INTERFACE I_RecipesManager

PROPERTY Active : REFERENCE TO BOOL
GET
END_GET
END_PROPERTY

PROPERTY Busy : REFERENCE TO BOOL
GET
END_GET
END_PROPERTY

PROPERTY Error : REFERENCE TO BOOL
GET
END_GET
END_PROPERTY

PROPERTY ErrorID : REFERENCE TO DWORD
GET
END_GET
END_PROPERTY

PROPERTY LastResult : REFERENCE TO E_RecipesManagerReturns
GET
END_GET
END_PROPERTY

METHOD MR_Abort : BOOL
VAR_INPUT
END_VAR
END_METHOD

METHOD MR_Backup : BOOL
VAR_INPUT
	sRecipesDefinition		: STRING;
	sRecipeName				: STRING;
	sBackupStoragePath		: STRING;
END_VAR
END_METHOD

METHOD MR_Create : BOOL
VAR_INPUT
	sRecipesDefinition : STRING;
	sRecipeName : STRING;
END_VAR
END_METHOD

METHOD MR_GetRecipesNames : BOOL
VAR_INPUT
	sRecipesDefinition : STRING;
END_VAR
END_METHOD

METHOD MR_GetVariablesNames : BOOL
VAR_INPUT
	sRecipesDefinition	: STRING;
	sRecipeName : STRING;
END_VAR
END_METHOD

METHOD MR_GetVariableValues : BOOL
VAR_INPUT
	sRecipesDefinition	: STRING;
	sRecipeName : STRING;
END_VAR
END_METHOD

METHOD MR_Init : BOOL
VAR_INPUT
END_VAR
END_METHOD

METHOD MR_Load : BOOL
VAR_INPUT
	sRecipesDefinition : STRING;
	sRecipeName : STRING;
END_VAR
END_METHOD

METHOD MR_LoadAndWritte : BOOL
VAR_INPUT
	sRecipesDefinition : STRING;
	sRecipeName : STRING;
END_VAR
END_METHOD

METHOD MR_Read : BOOL
VAR_INPUT
	sRecipesDefinition : STRING;
	sRecipeName : STRING;
END_VAR
END_METHOD

METHOD MR_ReadAndSave : BOOL
VAR_INPUT
	sRecipesDefinition : STRING;
	sRecipeName : STRING;
END_VAR
END_METHOD

METHOD MR_Reload : BOOL
VAR_INPUT
	sRecipeName : STRING;
	sRecipesDefinition : STRING;
END_VAR
END_METHOD

METHOD MR_ReloadExternal : BOOL
VAR_INPUT
	sRecipeName 			: STRING;
	sRecipesDefinition 		: STRING;
	sBackupStoragePath		: STRING;
END_VAR
END_METHOD

METHOD MR_Remove : BOOL
VAR_INPUT
	sRecipesDefinition : STRING;
	sRecipeName : STRING;
END_VAR
END_METHOD

METHOD MR_Restore : BOOL
VAR_INPUT
	sRecipesDefinition		: STRING;
	sRecipeName				: STRING;
	sBackupStoragePath		: STRING;
END_VAR
END_METHOD

METHOD MR_Save : BOOL
VAR_INPUT
	sRecipesDefinition : STRING;
	sRecipeName : STRING;
END_VAR
END_METHOD

METHOD MR_Writte : BOOL
VAR_INPUT
	sRecipesDefinition : STRING;
	sRecipeName : STRING;
END_VAR
END_METHOD

PROPERTY RecipeCount : REFERENCE TO USINT
GET
END_GET
END_PROPERTY

PROPERTY RecipesDefinition : REFERENCE TO STRING
GET
END_GET
END_PROPERTY

PROPERTY RecipesNames : REFERENCE TO ARRAY [0..iMAX_NUMBER_OF_RECIPES-1] OF STRING;
GET
END_GET
END_PROPERTY

PROPERTY RecipeValues : REFERENCE TO ARRAY [0..iMAX_NUMBER_OF_VARIABLES_IN_RECIPES-1] OF STRING
//PROPERTY RecipeValues : ARRAY [0..iMAX_NUMBER_OF_VARIABLES_IN_RECIPES-1] OF STRING(iMAX_RECIPE_NAME_LENGTH)
GET
END_GET
END_PROPERTY

PROPERTY RecipeValuesAdr : REFERENCE TO ARRAY [0..iMAX_NUMBER_OF_VARIABLES_IN_RECIPES-1] OF PVOID
GET
END_GET
END_PROPERTY

PROPERTY State : REFERENCE TO E_RecipesManagerState
GET
END_GET
END_PROPERTY

END_INTERFACE

(* stored: Version 1.1.0.1, ProductVersion 3.1.4024.12
   Itf I_RecipesManager: Id {7057ab11-af6e-493b-a220-bacdaa49dd59}
   Property Active: Id {bde34ffa-12f4-441f-bfba-71bea6fd0582}
   Get Get: Id {a452c6a0-c1af-48e5-8757-18e3cb39c475}
   Property Busy: Id {2dbc07eb-4c85-4755-acbe-ca1801cb3f83}
   Get Get: Id {d26ab1c0-6b9d-49af-bbbd-0b54b6950fb7}
   Property Error: Id {ec370076-02c1-427f-a7ce-cb62e257789d}
   Get Get: Id {a9ce79e2-c27c-447c-998e-74b99fc5c116}
   Property ErrorID: Id {03b3d0ee-1c04-4bd9-b50d-78faf2801a0d}
   Get Get: Id {ea298f4c-66d0-461e-b068-87476e613f9d}
   Property LastResult: Id {55507853-eb3f-47b7-b0e1-64c1557b8964}
   Get Get: Id {18c11fad-d0e3-4436-bbad-db091799d30a}
   Method MR_Abort: Id {43f4a9d7-ae84-4930-8a83-d7c761d7d38d}
   Method MR_Backup: Id {350fc49e-7a42-4963-bc6d-f348542a3a23}
   Method MR_Create: Id {b5dff985-0c90-4514-93bd-d89e0ee3d55c}
   Method MR_GetRecipesNames: Id {6ce1affd-3f1a-4148-8497-bf69ebefc106}
   Method MR_GetVariablesNames: Id {09bd1110-0d7f-4454-b702-d9613ede0d46}
   Method MR_GetVariableValues: Id {56bd768d-00f4-4b37-a666-dca3d11247b0}
   Method MR_Init: Id {8c99939b-3aa8-430b-922d-c6a8def04fc5}
   Method MR_Load: Id {33dd0eef-0d22-4d14-91e9-fb84e2d2b2bb}
   Method MR_LoadAndWritte: Id {3a1f24e4-f3cb-4c1b-8476-9940286f8a7d}
   Method MR_Read: Id {0dcbd69b-957a-410e-87c7-32a8393e30da}
   Method MR_ReadAndSave: Id {f38a0646-f35f-4d4b-ae1f-4a651c3f1bf6}
   Method MR_Reload: Id {ab64d9cf-1188-48f3-88e6-3c7e32af5756}
   Method MR_ReloadExternal: Id {9d321bef-5019-41e9-9b83-3d92834843d9}
   Method MR_Remove: Id {8dd2a9ab-d7bb-43e1-b8ef-ca690b7e82c2}
   Method MR_Restore: Id {d0caff79-8d4e-44d4-a4da-fb4758229a0d}
   Method MR_Save: Id {d3c65dfa-ba19-4fce-964e-891e5e86a4d5}
   Method MR_Writte: Id {85beb7bb-768a-41c1-8d96-3cc9c0197717}
   Property RecipeCount: Id {8dea1c76-d94a-47af-afde-307495d64bbd}
   Get Get: Id {7cf6118e-a992-464a-9529-638210286c15}
   Property RecipesDefinition: Id {e79cb469-7eac-4b13-8c1a-aa1b5864dc10}
   Get Get: Id {1526d50a-e62d-4506-8ff8-46a658cc24a1}
   Property RecipesNames: Id {9fcb0d35-8fca-4128-b9b3-5fa195d7a347}
   Get Get: Id {62bdd0db-e7e7-41b3-8ae6-5ce4905d2572}
   Property RecipeValues: Id {9de71902-b78e-4d2c-b2e3-a5aa7a35b706}
   Get Get: Id {9a8113d5-a3d5-425f-b71c-feb9dcebd1fb}
   Property RecipeValuesAdr: Id {5097eb6d-4186-47c4-a693-6e422f4a2757}
   Get Get: Id {aab75d28-cfc1-471a-bf58-198081c94f52}
   Property State: Id {d0bbd71e-19aa-499f-a925-0a93e89e0e31}
   Get Get: Id {ad02ac49-3806-4666-9d7a-a55dfb73c03a} *)
